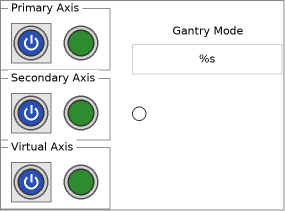
VISUALIZATION GantryControls  // 285x211
VAR_IN_OUT
	Gantry	:	HOMS_Gantry;
END_VAR
    GroupBox (0,0 110x70), "Primary Axis"
        PowerSwitch (11,23 40x40), variable: Gantry.PAxis.xEnable, behaviour: TOGGLE, style: Switch-PowerSwitch-Blue
        Lamp1 (61,23 40x40), variable: NOT Gantry.PAxis.stAxis.Status.Disabled, style: Lamp-Lamp1-Green
    GroupBox (0,70 110x70), "Secondary Axis"
        PowerSwitch (11,23 40x40), variable: Gantry.SAxis.xEnable, behaviour: TOGGLE, style: Switch-PowerSwitch-Blue
        Lamp1 (61,23 40x40), variable: NOT Gantry.SAxis.stAxis.Status.Disabled, style: Lamp-Lamp1-Green
    Textfield (132,44 150x30), "%s", text variable: Gantry.Mode
    Label (133,16 150x30), "Gantry Mode"
    RadioButton (130,82 150x63), variable: Gantry.ModeReq, input disabled if: Gantry.PAxis.stAxis.Status.Moving
        Areas[0]: Text=Coupled
        Areas[1]: Text=Decoupled
    GroupBox (0,139 110x70), "Virtual Axis", tooltip "For controlling coupled movement"
        PowerSwitch (11,23 40x40), variable: Gantry.VAxis.xEnable, behaviour: TOGGLE, style: Switch-PowerSwitch-Blue
        Lamp1 (61,23 40x40), variable: Gantry.SAxis.stAxis.Status.Coupled AND NOT Gantry.PAxis.stAxis.Status.Disabled AND NOT Gantry.SAxis.stAxis.Status.Disabled, style: Lamp-Lamp1-Green
END_VISUALIZATION

(* stored: Version 1.1.0.1, ProductVersion 3.1.4020.12
   Visu GantryControls: Id {94c9a656-b0ea-44da-b7d8-a5b59824712a} *)
